(*
Matrix Base Class
=============

Overview
-------------

This abstract class encapsulates the logic of manipulating and interacting with matricies without forcing a specific memory management pattern.
Derived classes are:

- DynamicMatrix: A concrete class that dynamically allocates memory to take any form needed
- StaticMatrix: An abstract class that serves as the base for classes with fixed memory sources
- MatrixAccessor: An abstract class that serves as the base for classes that inherit the memory of another matrix and remap it to their own form
 
With either pattern the memory is accessed as a row-major 1D array of LREAL.

*)
{attribute 'reflection'}
{attribute 'no_assign'}
FUNCTION_BLOCK ABSTRACT Matrix
VAR_INPUT
END_VAR
VAR_OUTPUT
END_VAR
VAR

	
	{attribute 'instance-path'}
	{attribute 'noinit'}
	sPath_ : T_MaxString;
	
	Ri : UINT;
	Ci : UINT;
	I : UINT;
	
	ZeroReference_ : LREAL;//numbers below this are considered zero for the purposes of avoiding near-divide-by-zero floating point issues
END_VAR

LogMessage('%s: There is no need to call the main FB function for type Matrix');

//returns the average value of all elements
PROPERTY PUBLIC Average : LREAL
GET
IF Length > 0 THEN
	Average := Sum / Length;
ELSE
	Average := 0;
END_IF
END_GET
END_PROPERTY

//The length (in Bytes) of the memory allocated to storing element data for this matrix
PROPERTY PUBLIC BufferSize : UDINT
GET
BufferSize := SIZEOF(LREAL)*Length;
END_GET
END_PROPERTY

//Resets the value of every element in this matrix to zero
METHOD PUBLIC Clear
VAR_INPUT
END_VAR
FillTrapezoidal(0,0,0);
END_METHOD

//Total number of columns in this matrix
PROPERTY PUBLIC ABSTRACT Cols : UINT
GET
END_GET
END_PROPERTY

(*Copy the value from each element in the source matrix to each corresponding element in this matrix

:Prerequisites:
 - This matrix is the same size as the source matrix
 - Neither matrix is empty
 
 *)
METHOD PUBLIC CopyFrom : BOOL//Returns true if the prerequisites were met and the data was copied, false otherwise
VAR_INPUT
	M : REFERENCE TO Matrix;//Source of the copy operation
END_VAR
CopyFrom := Matrix_Copy(M,THIS^);
END_METHOD

(*Copy the value from each element in this matrix to each corresponding element in the destination matrix

:Prerequisites:
 - This matrix is the same size as the destination matrix
 - Neither matrix is empty
 
 *)
METHOD PUBLIC CopyTo : BOOL//Returns true if the prerequisites were met and the data was copied, false otherwise
VAR_INPUT
	M : REFERENCE TO Matrix;//Destination for the copy operation
END_VAR
CopyTo := Matrix_Copy(THIS^,M);
END_METHOD

(*
For every element that exist in both this matrix and the source matrix, copy the value from the source matrix into this matrix
*)
METHOD PUBLIC FillFrom
VAR_INPUT
	M : REFERENCE TO Matrix;//source matrix for element copy operation
END_VAR
IF M.IsEmpty OR IsEmpty THEN
	RETURN;//no need to fill to/from empty matricies, and it
END_IF

FOR Ri := 0 TO MIN(Rows,M.Rows)-1 DO
	FOR Ci := 0 TO MIN(Cols,M.Cols)-1 DO
		SetRC(Ri,Ci,M.GetRC(Ri,Ci));
	END_FOR
END_FOR
END_METHOD

//Consider the subset of elements in this matrix starting and the supplied initial row and column as a submatrix. 
//For every element that exists in both the submatrix and the supplies source matrix, copy the value from the source matrix into the corresponding element of the submatrix.
METHOD PUBLIC FillFromAt
VAR_INPUT
	M : REFERENCE TO Matrix;//Source matrix for the copy operation
	RStart : UINT;//Row within this matrix to start the fill operation
	CStart : UINT;//Column within this matrix to start the fill operation
END_VAR
VAR
	SubMatrix : SubMatrixAccessor;
END_VAR
IF M.IsEmpty THEN
	LogWarning('%s: Attempt to fill from an empty matrix');
	RETURN;
END_IF

IF IsEmpty THEN
	LogWarning('%s: Attempt to fill into an empty matrix');
	RETURN;
END_IF

IF RStart >= Rows THEN
	LogWarning('%s: Attempt to fill out of bounds row of matrix');
	RETURN;
END_IF

IF CStart >= Cols THEN
	LogWarning('%s: Attempt to fill out of bounds col of matrix');
	RETURN;
END_IF

SubMatrix := M.GetSubMatrixAccessor(RStart,Rows-Rstart,CStart,Cols-CStart);
SubMatrix.FillFrom(M);
END_METHOD

//Fills all elements of this matrix based on which of three zones it is located into when considered as a trapezoidal matrix
METHOD PUBLIC FillTrapezoidal
VAR_INPUT
	Diagonal : LREAL;//Every element on the main diagonal of the matrix is set to this value.
	UpperRight : LREAL;//Every element above or to the right of the main diagonal is set to this value;
	LowerLeft : LREAL;//Every element below or to the left of the main diagonal is set to this value;
END_VAR
IF IsEmpty THEN
	LogWarning('%s: Attempt to trapezoid fill an empty matrix');
	RETURN;
END_IF


FOR Ri := 0 TO Rows-1 DO
	FOR Ci := 0 TO Cols-1 DO
		IF Ri = Ci THEN
			SetRC(Ri,Ci,Diagonal);
		ELSIF Ri < Ci THEN
			SetRC(Ri,Ci,UpperRight);
		ELSE
			SetRC(Ri,Ci,LowerLeft);
		END_IF
	END_FOR
END_FOR
END_METHOD

//Gets the determinant of this matrix
//
//:Prerequisites:
// - Matrix is not empty
// - Matrix is square
//
//.. note:: If this matrix does not meet the requirements 0 is returned
METHOD PUBLIC GetDeterminant : LREAL//The determinant of this matrix, if the prerequisites are met. Otherwise, returns 0.
VAR_INPUT
END_VAR
VAR
	Res : LREAL;
END_VAR
IF NOT(Matrix_Determinate(M := THIS^,Res => Res)) THEN
	LogWarning('%s: Unable to calculate determinate');
	GetDeterminant := 0;
ELSE
	GetDeterminant := Res;
END_IF
END_METHOD

//Gets the value of the element in this matrix at the supplied location as if the elements were stored in a 1D row-major array
//
//:Prerequisites:
// - I < Rows*Cols
// - Matrix is not empty
//
//.. note:: If the supplied index is out of bounds the value 0 is returned and a warning is generated in the Error List
METHOD PUBLIC ABSTRACT GetI : LREAL//The value of the element at the specified index, or 0 if an invalid index is supplied
VAR_INPUT
	I : UINT;//The index of the element which should have its value returned
END_VAR
END_METHOD

//returns the value of the element of this matrix at the specified row and column.
//
//:Prerequisites:
// - Row < Rows
// - Col < Cols
// - Matrix is not empty
//
//.. note:: If the supplied or or column is out of bounds then a warning message is generated in the Error List and the value 0 is returned
METHOD PUBLIC GetRC : LREAL//The value of the element at the specified row and column, or 0 if an invalid index is supplied
VAR_INPUT
	Row : UINT;//The row of the element to fetch
	Col : UINT;//The column of the element to fetch
END_VAR
IF IsEmpty THEN
	GetRC := 0;
	LogWarning('%s: Attempted RC access of empty Matrix');
ELSIF
	Row >= Rows THEN
	GetRC := 0;
	LogWarning('%s: Attempted RC access of out-of-bound matrix row');
ELSIF
	Col >= Cols THEN
	GetRC := 0;
	LogWarning('%s: Attempted RC access of out-of-bounds Matrix column');
ELSE
	GetRC := GetI(RC2I(Row,Col));
END_IF
END_METHOD

METHOD PUBLIC GetShrunkMatrixAccessor : ShrunkMatrixAccessor
VAR_INPUT
	Row : UINT;
	Col : UINT;
END_VAR
GetShrunkMatrixAccessor.Init(THIS^,Row,Col);
END_METHOD

//Returns the length of the matrix in the specified dimension
//
// - GetSize(0) is equivalent to Rows
// - GetSize(1) is equivalent to Cols
//
//.. note:: If an invalid dimension is supplied then a warning is generated in the Error List and the value 0 is returned
METHOD PUBLIC GetSize : UINT//The length of the matrix in the specified dimension, or 0 if the dimension specified is invalid
VAR_INPUT
	Dim : UINT;//The dimension of the matrix for which the size should be returned. 0=Rows, 1=Cols
END_VAR
IF Dim = 0 THEN
	GetSize := Rows;
ELSIF Dim = 1 THEN
	GetSize := Cols;
ELSE
	LogWarning('%s: Attempted to GetSize for a dimension other than 0 or 1');
	GetSize := 0;
END_IF
END_METHOD

//Calulates how long of a string (in Bytes) is required in order to print the entire contents of the matrix using the WriteDataToString function
METHOD PUBLIC GetStringLengthEstimate : UDINT;
VAR_INPUT
END_VAR
VAR
	CharsPerElement : UDINT := 20;//15 point precision, decimal, sign, leading zero, comma, space
	CharsPerRow : UDINT := 6;//space, semicolon, carriage return, line return, space, space
	CharsPerMatrix : UDINT := 4;//open bracket, space ; space, closing bracket
END_VAR
GetStringLengthEstimate := 1+CharsPerMatrix + CharsPerRow * Rows + CharsPerElement * Length;//extra one for null character
END_METHOD

METHOD PUBLIC GetSubMatrixAccessor : SubMatrixAccessor
VAR_INPUT
	RowStart : UINT;
	RowCount : UINT;
	ColStart : UINT;
	ColCount : UINT;
END_VAR
GetSubMatrixAccessor.Init(THIS^,RowStart,RowCount,ColStart,ColCount);
END_METHOD

METHOD PUBLIC GetTransposeMatrixAccessor : TransposeMatrixAccessor
VAR_INPUT
END_VAR
GetTransposeMatrixAccessor.Init(THIS^);
END_METHOD

//Returns the vector dot product of this matrix and the supplied other matrix (ignoring the orientation of both matricies).
//:Prerequisites:
// - This matrix is a vector and is not empty
// - The supplied other matrix is a vector and is not empty
// - This vector has the same length (but not necessarily orientation) as the supplied vector
METHOD PUBLIC GetVectorDotProduct : LREAL//The dot product (element-wise product) of this vector and the supplied vector, or 0 if the inputs are invalid
VAR_INPUT
	V : REFERENCE TO Matrix;//The vector which which the dot product of this vector should be taken.
END_VAR
VAR
	Res : LREAL;
END_VAR
IF NOT(Vector_DotProduct(V,THIS^,Res => Res)) THEN
	LogWarning('%s: Unable to calculate vector dot product');
	GetVectorDotProduct := 0;
ELSE
	GetVectorDotProduct := Res;
END_IF
END_METHOD

//Calcualtes the vector magnitude of this matrix (square root of the sum of the squares), assuming it is a vector.
//
//:Prerequisites:
// - This matrix is not empty and is a vector
//
//.. note:: If this matrix is empty or is not a vector, 0 is returned
METHOD PUBLIC GetVectorMagnitude : LREAL//The vector magnitude of this matrix if it is a vector, otherwise 0
VAR_INPUT
END_VAR
VAR
	Res : LREAL;
END_VAR
IF NOT(Vector_Magnitude(THIS^,Res => Res)) THEN
	LogWarning('%s: Unable to calculate vector magnitude');
	GetVectorMagnitude := 0;
ELSE
	GetVectorMagnitude := Res;
END_IF
END_METHOD

METHOD PROTECTED IC2RC
VAR_INPUT
	Index : UINT;
	ColCount : UINT;
END_VAR
VAR_OUTPUT
	Row : UINT;
	Col : UINT;
END_VAR
Col := Index MOD ColCount;
Row := (Index - Col) / ColCount;
END_METHOD

//Raises every element of the matrix to the supplied power
METHOD PUBLIC IntPower
VAR_INPUT
	Exponent : INT;//Power with which to raise every element of the matrix
END_VAR
IF IsEmpty THEN
	RETURN;
END_IF
FOR I := 0 TO Length-1 DO
	SetI(I,EXPT(GetI(I),Exponent));
END_FOR
END_METHOD

//Returns true if the matrix does not have any addresible elements
PROPERTY PUBLIC IsEmpty : Bool
GET
IsEmpty := Length = 0;
END_GET
END_PROPERTY

//Determines if this matrix is equal to a supplied matrix.
//
//Two matricies are considered equal if they are the same size and every set of corresponding elements are equal.
//
//.. note:: Two empty matricies are considered equal.
METHOD PUBLIC IsEqual : BOOL//TRUE if the two matricies are equal, FALSE if they are not
VAR_INPUT
	M : REFERENCE TO Matrix;//The other matrix to compare to this one
END_VAR
IF NOT( IsEqualSize(M)) THEN
	IsEqual := FALSE;
	RETURN;
END_IF

//If either matrix is empty don't bother comparing elements
IF IsEmpty OR M.IsEmpty THEN
	//If both are empty then they are equal
	IsEqual := IsEmpty AND M.IsEmpty;
	RETURN;
END_IF

//Both Rows and Cols must be non zero for this loop to not go bonkers
FOR Ri := 0 TO Rows-1 DO
	FOR Ci := 0 TO Cols-1 DO
		IF NOT(GetRC(Ri,Ci) = M.GetRC(Ri,Ci)) THEN
			IsEqual := FALSE;
			RETURN;
		END_IF
	END_FOR
END_FOR

IsEqual := TRUE;
END_METHOD

//Checks if this matrix is the same size (number of rows and number of columns match) as the supplied matrix.
//
//.. note:: two empty matricies are considered the same size.
METHOD PUBLIC IsEqualSize : BOOL//True if this matrix is the same size as the supplied matrix
VAR_INPUT
	M : REFERENCE TO Matrix;//The matrix which should have its size compared to the size of this matrix
END_VAR
IsEqualSize := M.Rows = Rows AND M.Cols = Cols;
END_METHOD

//Determines if this matrix is *nearly* equal to a supplied matrix, based on a supplied precision.
//
//Two matricies are considered nearly equal if they are the same size and every set of corresponding elements are equal to within the supplied precision.
//.. note:: Note that two empty matricies are considered equal
METHOD PUBLIC IsNearlyEqual : BOOL//TRUE if the two matricies are nearly equal, FALSE if they are not
VAR_INPUT
	M : REFERENCE TO Matrix;//The other matrix to compare to this one
	Precision : LREAL;//Deviation between two elements larger than this value makes them unequal
END_VAR
IF NOT( IsEqualSize(M)) THEN
	IsNearlyEqual := FALSE;
	RETURN;
END_IF

//If either matrix is empty don't bother comparing elements
IF IsEmpty OR M.IsEmpty THEN
	//If both are empty then they are equal
	IsNearlyEqual := IsEmpty AND M.IsEmpty;
	RETURN;
END_IF

//Both Rows and Cols must be non zero for this loop to not go bonkers
FOR Ri := 0 TO Rows-1 DO
	FOR Ci := 0 TO Cols-1 DO
		IF NOT( ABS(GetRC(Ri,Ci) - M.GetRC(Ri,Ci)) < Precision) THEN
			IsNearlyEqual := FALSE;
			RETURN;
		END_IF
	END_FOR
END_FOR

IsNearlyEqual := TRUE;
END_METHOD

//Returns true if the supplied value is near enough to zero that it should not be used as a divisor. See the property ZeroReference
METHOD PROTECTED IsNearZero : BOOL
VAR_INPUT
	IN : LREAL;//The value which should have its magnitude evaluated
END_VAR
IsNearZero := ABS(IN) < ZeroReference;
END_METHOD

//Returns true if this matrix is not empty, and the number of columns is equal to the number of rows
PROPERTY PUBLIC IsSquare : BOOL
GET
IsSquare := NOT(IsEmpty) AND Rows = Cols;
END_GET
END_PROPERTY

//Returns true if this matrix is not empty, and at least one dimension has a size of 1 (row vector or column vector).
PROPERTY PUBLIC IsVector : BOOL
GET
IsVector := NOT(IsEmpty) AND (Rows = 1) OR (Cols = 1);
END_GET
END_PROPERTY

//Total number of elements in this matrix
PROPERTY PUBLIC Length : UINT
GET
Length := Rows * Cols;
END_GET
END_PROPERTY

//Logs the supplied message to the error output as an 'Error'
METHOD PROTECTED LogError
VAR_INPUT
	Message : T_MaxString;//The message to log. %s is substituted with the symbolic address of this matrix.
END_VAR
ADSLOGSTR(ADSLOG_MSGTYPE_WARN,Message,sPath);
END_METHOD

//Logs the supplied message to the windoes event log
METHOD PROTECTED LogEvent
VAR_INPUT
	Message : T_MaxString;//The message to log. %s is substituted with the symbolic address of this matrix.
END_VAR
ADSLOGSTR(ADSLOG_MSGTYPE_LOG,Message,sPath);
END_METHOD

//Logs the supplied message to the error output as a 'Message'
METHOD PROTECTED LogMessage
VAR_INPUT
	Message : T_MaxString;//The message to log. %s is substituted with the symbolic address of this matrix.
END_VAR
ADSLOGSTR(ADSLOG_MSGTYPE_STRING,Message,sPath);
END_METHOD

//Logs the supplied message to the error output as a 'Warning'
METHOD PROTECTED LogWarning
VAR_INPUT
	Message : T_MaxString;//The message to log. %s is substituted with the symbolic address of this matrix.
END_VAR
ADSLOGSTR(ADSLOG_MSGTYPE_WARN,Message,sPath);
END_METHOD

//Returns the maximum value from all elements
PROPERTY PUBLIC MaxVal : LREAL
GET
VAR
	MaxVal_ : LREAL;
END_VAR
IF IsEmpty THEN
	MaxVal := 0;
ELSE
	MaxVal_ := GetI(0);
	FOR I := 1 TO Length-1 DO
		IF getI(I) < MaxVal_ THEN
			MaxVal_ := GetI(I);
		END_IF
	END_FOR
	MaxVal := MaxVal_;
END_IF
END_GET
END_PROPERTY

//Returns the minimum value from all elements
PROPERTY PUBLIC MinVal : LREAL
GET
VAR
	MinVal_ : LREAL;
END_VAR
IF IsEmpty THEN
	MinVal := 0;
ELSE
	MinVal_ := GetI(0);
	FOR I := 1 TO Length-1 DO
		IF getI(I) < MinVal_ THEN
			MinVal_ := GetI(I);
		END_IF
	END_FOR
	MinVal := MinVal_;
END_IF
END_GET
END_PROPERTY

//Scales every element of the matrix by the inverse of the magnitude.
//
// - Vector magnitude is determined by GetVectorMagnitude
// - Square Matrix magnitude is determined by GetDeterminate
// - Rectangular matricies produce an error
//
//:Prerequisites: 
// - matrix is not empty
// - matrix is not rectangular
METHOD PUBLIC Normalize : BOOL//TRUE if the matrix was normalized. FALSE if not.
VAR_INPUT
END_VAR
VAR
	Mag : LREAL;
END_VAR
VAR CONSTANT
	
END_VAR
IF IsEmpty THEN
	Normalize := FALSE;
	LogWarning('%s: Unable to normalize matrix because it is empty');
	RETURN;
ELSIF IsVector THEN
	Mag := GetVectorMagnitude();
ELSIF IsSquare THEN
	Mag := GetDeterminant();
ELSE
	Normalize := FALSE;
	LogWarning('%s: Unable to normalize matrix because it is not square or a vector');
	RETURN;
END_IF

IF IsNearZero(Mag) THEN
	Normalize := FALSE;
	LogWarning('%s: Unable to normalize matrix because the magnitude was too close to zero');
	RETURN;
END_IF

Normalize := TRUE;

Scale(1/Mag);
END_METHOD

//Raises every element of the matrix to the supplied power
//
//.. caution:: Many values of exponent could easily cause all of the elements to turn into NaN!
METHOD PUBLIC Power
VAR_INPUT
	Exponent : LREAL;//Power with which to raise every element of the matrix
END_VAR
IF IsEmpty THEN
	RETURN;
END_IF
FOR I := 0 TO Length-1 DO
	SetI(I,EXPT(GetI(I),Exponent));
END_FOR
END_METHOD

//Computes the index in a row-major 1D array representing this Matrix given a supplied Row and Column index
METHOD PROTECTED RC2I : UINT//The 0-based index of the element in the 1D array
VAR_INPUT
	Row : UINT;//The target row of the element
	Col : UINT;//The target column of the element
END_VAR
RC2I := RCC2I(Row,Col,Cols);
END_METHOD

//Computes the index in a row-major 1D array representing a Matrix with the supplied number of columns (*NOT this matrix*) given a supplied Row and Column index
METHOD PROTECTED RCC2I : UINT//Index of the element in a 1D array
VAR_INPUT
	Row : UINT;//Row of the target element
	Col : UINT;//Column fo the target element
	ColCount : UINT;//The number of columns in the 1D array (not necessarilly the number of columns in this Matrix!)
END_VAR
RCC2I := Row*ColCount + Col;
END_METHOD

//Total number of rows in this matrix
PROPERTY PUBLIC ABSTRACT Rows : UINT
GET
END_GET
END_PROPERTY

//Scales every element of this matrix by the supplied value.
METHOD PUBLIC Scale
VAR_INPUT
	Scalar : LREAL;//Value with which to scale every element of this matrix
END_VAR
Matrix_Scale(THIS^,Scalar);
END_METHOD

//Sets the element specified by the supplied index to the suppleid value, assuming the data of the matrix is stored in a 1D row-major array
//
//:Prerequisites: - I < Rows*Cols
METHOD PUBLIC ABSTRACT SetI : BOOL//TRUE if the specified index is valid and the data is copied. FLASE otherwise
VAR_INPUT
	I : UINT;//The index specifying which element should be modified
	Val : LREAL;//The value copied to the corresponding element
END_VAR
END_METHOD

//Sets the element specified by the supplied row and column to the suppleid value
//
//:Prerequisites:
// - Row < Rows
// - Col < Cols
METHOD PUBLIC SetRC : BOOL;//TRUE if the specified row and column are valid and the data is copied. FALSE otherwise
VAR_INPUT
	Row : UINT;//The row of the element to set
	Col : UINT;//The column of the element to set
	Val : LREAL;//The value to copy into the specified element
END_VAR
IF IsEmpty THEN
	SetRC := FALSE;
	LogWarning('%s: Attempt to set data using RC access when data is not initialized');
ELSIF Row >= Rows THEN
	SetRC := FALSE;
	LogWarning('%s: Attempt to set data using RC access when Row is out of bounds');
ELSIF Col >= Cols THEN
	SetRC := FALSE;
	LogWarning('%s: Attempt to set data using RC access when Col is out of bounds');
ELSE
	SetRC := SetI(RC2I(Row,Col),Val);
END_IF
END_METHOD

//The symbolic path to this matrix in memory
PROPERTY PUBLIC sPath : T_MaxString
GET
sPath := sPath_;
END_GET
END_PROPERTY

//Returns the sum of all elements
PROPERTY PUBLIC Sum : LREAL
GET
VAR
	Sum_ : LREAL;
END_VAR
Sum_ := 0;
IF NOT(IsEmpty) THEN
	FOR I := 0 TO Length-1 DO
		Sum_ := Sum_ + GetI(I);
	END_FOR
END_IF
Sum := Sum_;
END_GET
END_PROPERTY

//Writes the elements of this matrix to a string in a human-readable way, up to the specified length.
//
//Use the GetStringLengthEstimate function to calculate how much memory is necessary to output the entire matrix to one string
METHOD PUBLIC WriteDataToString : BOOL//Returns true if the entire matrix was written to the string, false otherwise
VAR_INPUT
	Buffer : POINTER TO STRING;//The output buffer that should be overwritten with the contents of the matrix
	BufferLen : UDINT;//The length, in bytes, of the output buffer available fo writing
END_VAR
VAR
	Temp : STRING(32);
	Pos : UDINT;
END_VAR
VAR CONSTANT
	ColSep : STRING(2) := ', ';
	RowSep : STRING(6) := ' ;$R$L  ';
	MatStart : STRING(2) := '[ ';
	MatEnd : STRING(2) := ' ]';
END_VAR
Pos := 0;
IF NOT(STRNCPY(Buffer+Pos,ADR(MatStart),BufferLen-Pos)) THEN
	WriteDataToString := FALSE;
	RETURN;
END_IF;
Pos := Pos + LEN2(ADR(MatStart));

FOR Ri := 0 TO Rows-1 DO
	IF Ri <> 0 THEN
		IF NOT(STRNCPY(Buffer+Pos,ADR(RowSep),BufferLen-Pos)) THEN
			WriteDataToString := FALSE;
			RETURN;
		END_IF;
		Pos := Pos + LEN2(ADR(RowSep));
	END_IF;

	FOR Ci := 0 TO Cols-1 DO
		IF Ci <> 0 THEN
			IF NOT(STRNCPY(Buffer+Pos,ADR(ColSep),BufferLen-Pos)) THEN
				WriteDataToString := FALSE;
				RETURN;
			END_IF;
			Pos := Pos + LEN2(ADR(ColSep));
		END_IF;
		
		Temp := LREAL_TO_STRING(GetRC(Ri,Ci));
		IF NOT(STRNCPY(Buffer+Pos,ADR(Temp),BufferLen-Pos)) THEN
			WriteDataToString := FALSE;
			RETURN;
		END_IF;
		Pos := Pos + LEN2(ADR(Temp));
	END_FOR
END_FOR

IF NOT(STRNCPY(Buffer+Pos,ADR(MatEnd),BufferLen-Pos)) THEN
	WriteDataToString := FALSE;
	RETURN;
END_IF;
Pos := Pos + LEN2(ADR(MatEnd));
WriteDataToString := TRUE;
END_METHOD

//Values with a magnitude lower than this value will be considered as zero for purposes of avoiding divide by zero errors
PROPERTY PUBLIC ZeroReference : LREAL
GET
ZeroReference := ZeroReference_;
END_GET
SET
ZeroReference_ := ZeroReference;
END_SET
END_PROPERTY

END_FUNCTION_BLOCK

(* stored: Version 1.1.0.1, ProductVersion 3.1.4024.9
   POU Matrix: Id {37681762-a9e8-4dd1-b97b-ca342c51c659}, SpecialFunc None
   Folder Accessors: Id {ef6a5473-da01-0d79-286e-6646d04a6f5a}
   Folder Aggregators: Id {c541bfa3-492b-0df6-1926-f02606816bce}
   Folder Comparators: Id {b7fe62c6-6f13-454d-9f2a-eae01884c717}
   Folder Getters: Id {764d70ab-da43-41bc-a172-c1370fa4e2a7}
   Folder Helpers: Id {c18f9319-b519-4a83-98b2-43ca8f72caca}
   Folder Modifiers: Id {0b7b615a-d2d6-4e62-b148-1a83ef247c62}
   Folder Properties: Id {63bcd68f-51b7-4cdd-bc76-abfb7c04d216}
   Folder Protected: Id {52ab6c01-12bf-4ee4-b7d8-7459de792de0}
   Property Average: Id {bbb5565e-c8b8-06a4-072f-2f69a4299899}
   Get Get: Id {3df0d655-ce9c-0473-3f0c-ac0787664407}
   Property BufferSize: Id {f271d29f-8d22-4870-9606-910840251c4c}
   Get Get: Id {cde88b07-59bd-48ab-b6be-612e25f0f9b5}
   Method Clear: Id {788b000b-9652-4513-87ea-afa0efbc93b4}
   Property Cols: Id {d523fd23-40b0-0c12-048f-35d989fa4f45}
   Get Get: Id {a7a6e0d6-1627-0349-3c56-d4f322f68321}
   Method CopyFrom: Id {dae02926-a792-0e0c-1dd5-5763605fc7fb}
   Method CopyTo: Id {8ef25dfb-afc0-053f-1591-86389e6847af}
   Method FillFrom: Id {022b237b-0584-4ce7-a547-77e65ab3d048}
   Method FillFromAt: Id {57397ef9-06ec-050d-1f21-ec905dd7b0ad}
   Method FillTrapezoidal: Id {f5fa3a45-37d2-08ef-0015-41ed1be8ef4b}
   Method GetDeterminant: Id {4690878e-585c-49dd-a170-b0f3c7ff17f5}
   Method GetI: Id {15777527-77a2-42cc-8d9c-f624271cdfcd}
   Method GetRC: Id {fa44f9d9-95b5-4fc6-badf-738b5a3911f1}
   Method GetShrunkMatrixAccessor: Id {a17e9bb7-2275-05d1-18ac-48a4fa653049}
   Method GetSize: Id {61a33f57-364a-4e27-9ba3-9caf9ad98b8f}
   Method GetStringLengthEstimate: Id {105d6985-ce7b-0363-01e4-eb441c24368f}
   Method GetSubMatrixAccessor: Id {a144ad62-4358-0927-0b6b-026cfc4aa1d5}
   Method GetTransposeMatrixAccessor: Id {5dc6f40a-ecba-0ce5-0744-b541aad5ef72}
   Method GetVectorDotProduct: Id {1658fad0-9792-0d13-3da1-4022c6478285}
   Method GetVectorMagnitude: Id {2cda7f0d-36ea-0716-0a39-1b669b254390}
   Method IC2RC: Id {7255f7df-750d-0f66-22e3-0b875b59a237}
   Method IntPower: Id {6bdcc943-6222-00fa-3a06-a537022f40c0}
   Property IsEmpty: Id {c235a1c3-19da-47f7-9309-34932eb65324}
   Get Get: Id {ae4f7dd7-6afa-42b8-914f-506a87feabaa}
   Method IsEqual: Id {864b7d2e-c191-4c91-985a-939f8832c318}
   Method IsEqualSize: Id {27be0354-ccaa-4d4d-aa11-92c8ff0d05d2}
   Method IsNearlyEqual: Id {5d748479-c05b-0288-3d27-e100bad6055b}
   Method IsNearZero: Id {14d96c82-fff9-0250-2cd6-b017194a9777}
   Property IsSquare: Id {e672b3bd-9ada-4884-9298-de073113df9b}
   Get Get: Id {4255b8b2-db7d-4f6c-90fc-32930d8d75f2}
   Property IsVector: Id {fa53e68e-f9cd-4264-b4bc-c5aa3563b636}
   Get Get: Id {37d299d5-2a39-4c73-888a-5f06acc43d3e}
   Property Length: Id {2c497c08-f008-0342-1d0c-6819a4969e69}
   Get Get: Id {fc001511-17d0-03a1-3ade-ffcc96d39c1c}
   Method LogError: Id {0d93f53f-aa75-038c-24c9-4008df3d6da2}
   Method LogEvent: Id {8171c1d6-5906-0bfd-0ba5-b722be9c1e72}
   Method LogMessage: Id {97d8748b-f9e0-0605-025f-e9b0af536375}
   Method LogWarning: Id {9209617a-719a-05c3-2a97-800df97be0bd}
   Property MaxVal: Id {2e28b031-b417-0f4a-0152-01ef3cd1db57}
   Get Get: Id {f7bebe36-e3d7-072e-0310-06c7d57e73dc}
   Property MinVal: Id {02b2c522-52fd-07a2-0002-77487d44cc65}
   Get Get: Id {cbaba9d2-d69b-0140-2c06-09a756014561}
   Method Normalize: Id {404b4c10-5aeb-0370-10b6-f0f7c656ed69}
   Method Power: Id {554d7c44-e24f-0d64-3e72-fbca02a11c79}
   Method RC2I: Id {3fa58cb3-47e4-0750-1d7e-28cc355ab4a5}
   Method RCC2I: Id {a76e2565-d4ef-4b3c-baf9-76f94e292fe8}
   Property Rows: Id {d28429c0-8643-0547-1543-63793204cffa}
   Get Get: Id {38f7288d-05a9-0a44-1ad7-57f45d3df90f}
   Method Scale: Id {b7f3a516-3a74-41d5-8946-fd12d55e7c87}
   Method SetI: Id {1887d363-8acf-46d8-a10f-82241082042b}
   Method SetRC: Id {95b644b0-5978-469a-8c47-6f924bbad114}
   Property sPath: Id {71b212c0-e2af-08e9-0666-16cfb7faa00b}
   Get Get: Id {5efaf036-abb9-0591-2a9d-5c04faea0e41}
   Property Sum: Id {26264213-af04-0fe3-15b5-fce4debe5ded}
   Get Get: Id {98d20894-bd36-02b2-129d-e600f0a5d072}
   Method WriteDataToString: Id {7c9446a3-69a9-08e8-3b1c-3852339b4db4}
   Property ZeroReference: Id {c759c62c-8641-003b-19d2-c7e06780aedd}
   Get Get: Id {72e7fd1c-4821-0afe-1307-1af2cfef9288}
   Set Set: Id {b7e81f92-1be0-0ef9-012d-c2c5baa8b706} *)
